PROGRAM PRG_MachineControl
VAR
	bFirstCycle 		: BOOL := TRUE;			(*  *)
	fbMachineControler 	: FB_MachineControl;	(*  *)
	fbFileLogger 		: FB_FileLogger;		(*	*)
END_VAR

IF bFirstCycle THEN
	bFirstCycle := FALSE;
	
	(* Assign machine controler reference to Shell API*)
	stShell.stPlatform.ref_fbMachineControler REF= fbMachineControler;
	
	(* Set assignamnet done bit for visu controler *)
	stShell.stFlags.bMachineCtrlAssignamentsDone := TRUE;
	
	fbMachineLogger.MR_FirstCycle( 	sName		:= 'PSE_Shell_Machine_Logger',
									sFileDir 	:= 'C:\TwinCAT\Projects\Loggers',
									sFileName 	:= 'PSE_Shell_Machine_Logger',
									sAmsNetId 	:= '',
									bAddTimeStamp := FALSE,
									bAddHeader := FALSE);
END_IF

IF NOT fbMachineLogger.Active THEN 
	fbMachineLogger.MR_Init();	
END_IF

fbMachineTime(bEnable := TRUE);
fbMachineControler();
fbMachineLogger();

END_PROGRAM

(* stored: Version 1.1.0.1, ProductVersion 3.1.4024.9
   POU PRG_MachineControl: Id {060380e8-9f13-4409-a4b0-3cef7b843ba9}, SpecialFunc None *)
